DATA_BLOCK "ST10_PM"
{ S7_Optimized_Access := 'FALSE' }
VERSION : 0.1
   STRUCT
      Num { S7_SetPoint := 'False'} : Array[1..32] of "RCS_PMInterface_V1";
      Status { S7_SetPoint := 'True'} : Array[1..50] of Int;
   END_STRUCT;


BEGIN

END_DATA_BLOCK

